// SIMATIC S7-200 project (STEP 7-Micro/WIN), CPU 226 CN REL 02.01

SYMBOL_TABLE 变量
接收字节数            VB0
从站地址             VB1
保持寄存器起始地址        VD2
最大IO点数           VW6
最大AI通道数          VW8      // 可为16或32
保持寄存器数量          VW10
数据包合法性           V12.0    // 只有该位为1才会处理数据包
接收存储区            VB13
发送存储区            VB268
END_SYMBOL_TABLE

SYMBOL_TABLE Modbus地址
M0001            QB0      // 00001~00128
M10001           IB0      // I0.0~I15.7
M3000            AIW0     // AIW0~AIW62
END_SYMBOL_TABLE

ORGANIZATION_BLOCK 主程序:OB1
TITLE=程序注释
BEGIN
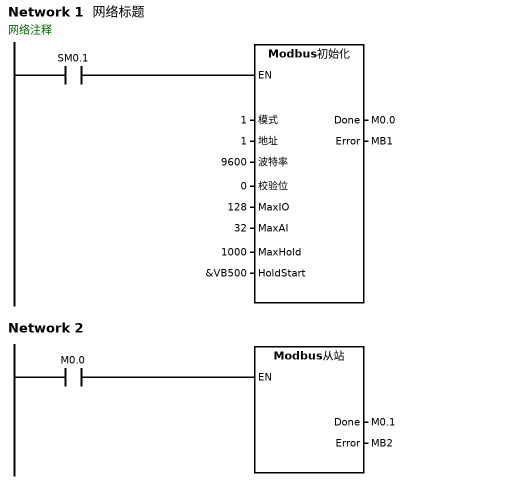
Network 1 // 网络标题
// 网络注释
LD     SM0.1
CALL   Modbus初始化:SBR0, 1, 1, 9600, 0, 128, 32, 1000, &VB500, M0.0, MB1
Network 2
LD     M0.0
CALL   Modbus从站:SBR1, M0.1, MB2
END_ORGANIZATION_BLOCK

SUBROUTINE_BLOCK Modbus初始化:SBR0
TITLE=此程序初始化Modbus所需参数
// 校验位:
// 0 - 无校验
// 1 - 奇校验
// 2 - 偶校验
// 
// Error值在Done位为0时有效
// Error值含义:
// 1 - 波特率初始化失败
// 2 - 校验位初始化失败
// 3 - 没有相关模式
VAR_INPUT
模式:BYTE;	// LB0 0 - 禁用Modbus库、1 - 启用Modbus库
地址:BYTE;	// LB1 从站地址
波特率:DWORD;	// LD2 通讯所需波特率
校验位:BYTE;	// LB6 数据包校验位
MaxIO:INT;	// LW7 
MaxAI:INT;	// LW9 可为16或32
MaxHold:INT;	// LW11 
HoldStart:DWORD;	// LD13 
END_VAR
VAR_OUTPUT
Done:BOOL;	// L17.0 0 - 初始化失败、1 - 初始化成功
Error:BYTE;	// LB18 
END_VAR
VAR
自由口控制:BYTE;	// LB19 
初始化标志:BYTE;	// LB20 
END_VAR
BEGIN
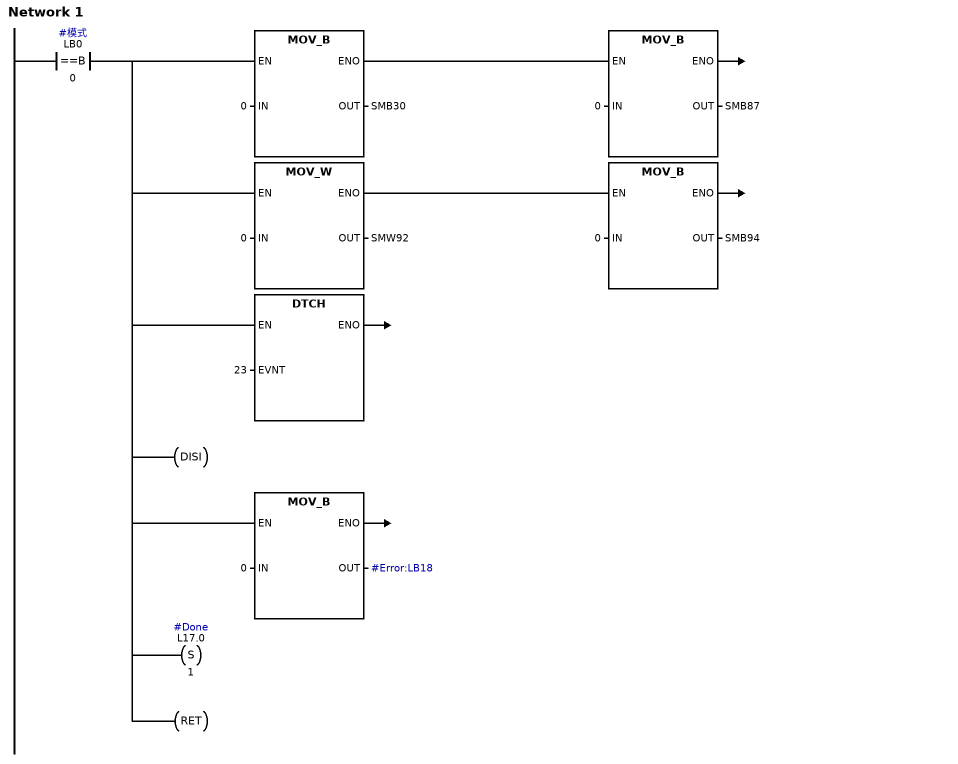
Network 1
LDB=   #模式:LB0, 0
LPS
MOVB   0, SMB30
AENO
MOVB   0, SMB87
LRD
MOVW   0, SMW92
AENO
MOVB   0, SMB94
LRD
DTCH   23
LRD
DISI
LRD
MOVB   0, #Error:LB18
LRD
S      #Done:L17.0, 1
LPP
CRET
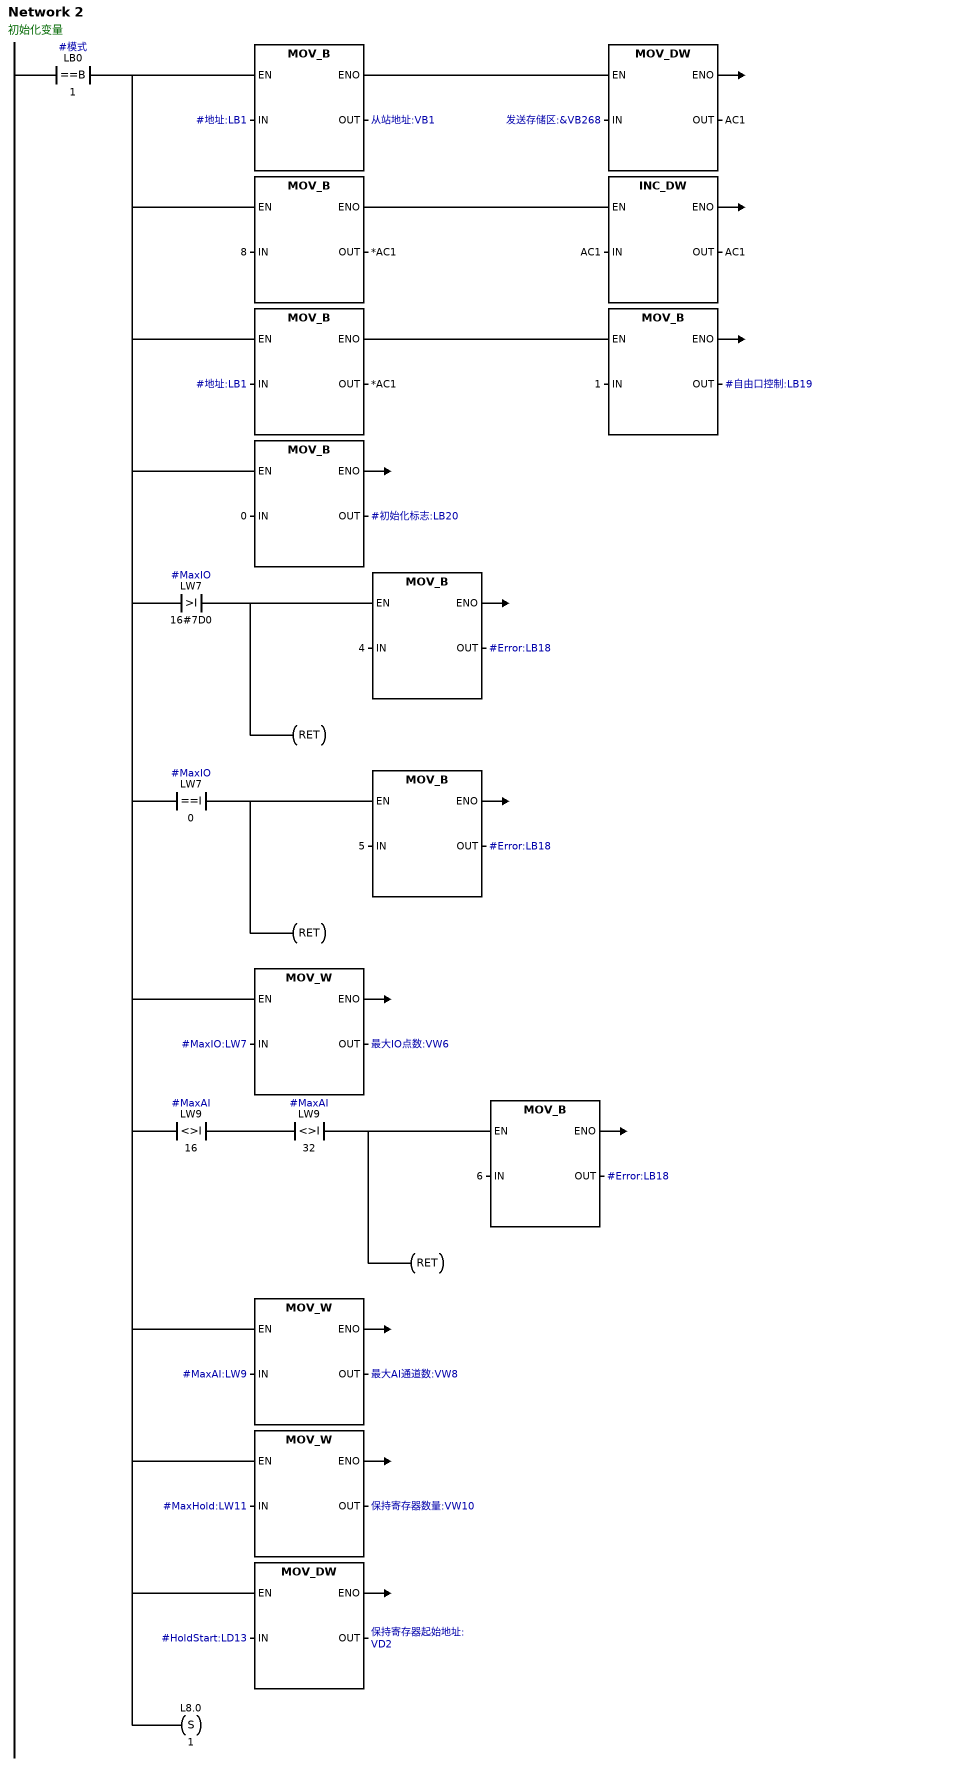
Network 2
// 初始化变量
LDB=   #模式:LB0, 1
LPS
MOVB   #地址:LB1, 从站地址:VB1
AENO
MOVD   &发送存储区:VB268, AC1
LRD
MOVB   8, *AC1
AENO
INCD   AC1
LRD
MOVB   #地址:LB1, *AC1
AENO
MOVB   1, #自由口控制:LB19
LRD
MOVB   0, #初始化标志:LB20
LRD
AW>    #MaxIO:LW7, 16#7D0
MOVB   4, #Error:LB18
CRET
LRD
AW=    #MaxIO:LW7, 0
MOVB   5, #Error:LB18
CRET
LRD
MOVW   #MaxIO:LW7, 最大IO点数:VW6
LRD
AW<>   #MaxAI:LW9, 16
AW<>   #MaxAI:LW9, 32
MOVB   6, #Error:LB18
CRET
LPP
MOVW   #MaxAI:LW9, 最大AI通道数:VW8
MOVW   #MaxHold:LW11, 保持寄存器数量:VW10
MOVD   #HoldStart:LD13, 保持寄存器起始地址:VD2
S      L8.0, 1
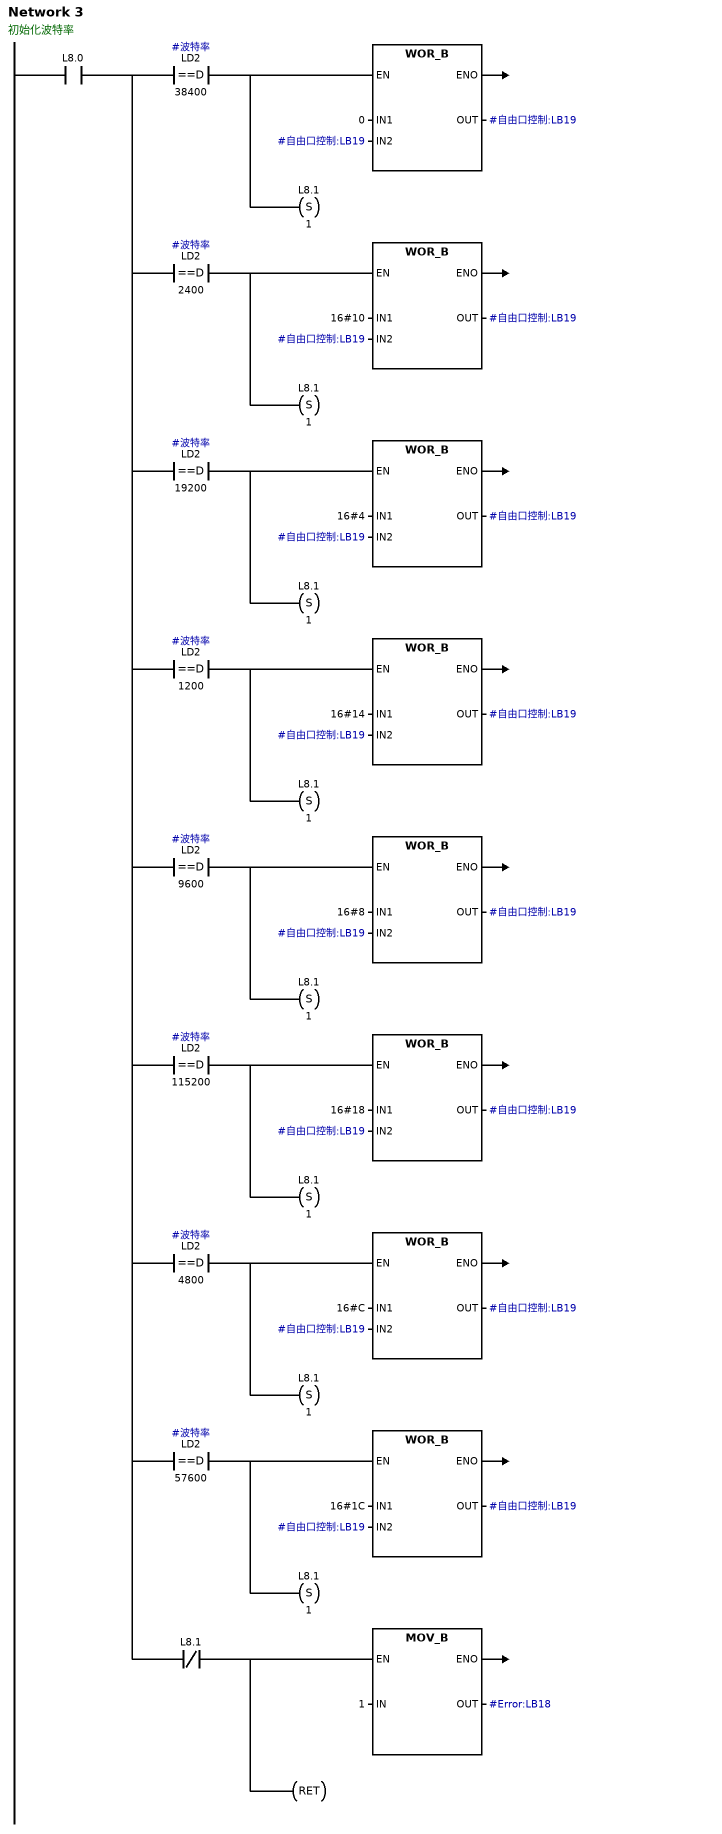
Network 3
// 初始化波特率
LD     L8.0
LPS
AD=    #波特率:LD2, 38400
ORB    0, #自由口控制:LB19
S      L8.1, 1
LRD
AD=    #波特率:LD2, 2400
ORB    16#10, #自由口控制:LB19
S      L8.1, 1
LRD
AD=    #波特率:LD2, 19200
ORB    16#4, #自由口控制:LB19
S      L8.1, 1
LRD
AD=    #波特率:LD2, 1200
ORB    16#14, #自由口控制:LB19
S      L8.1, 1
LRD
AD=    #波特率:LD2, 9600
ORB    16#8, #自由口控制:LB19
S      L8.1, 1
LRD
AD=    #波特率:LD2, 115200
ORB    16#18, #自由口控制:LB19
S      L8.1, 1
LRD
AD=    #波特率:LD2, 4800
ORB    16#C, #自由口控制:LB19
S      L8.1, 1
LRD
AD=    #波特率:LD2, 57600
ORB    16#1C, #自由口控制:LB19
S      L8.1, 1
LPP
AN     L8.1
MOVB   1, #Error:LB18
CRET
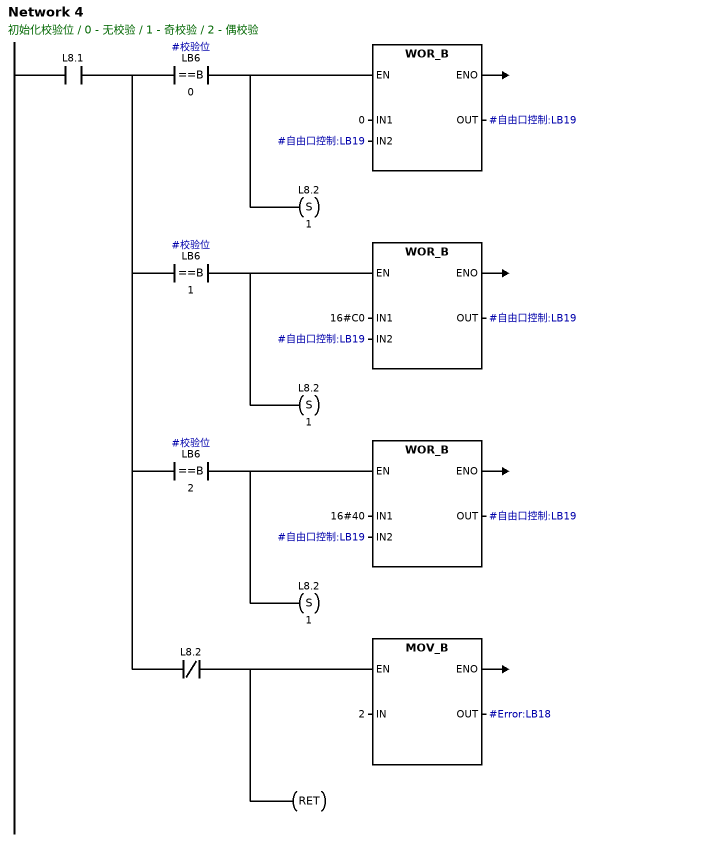
Network 4
// 初始化校验位
// 0 - 无校验
// 1 - 奇校验
// 2 - 偶校验
LD     L8.1
LPS
AB=    #校验位:LB6, 0
ORB    0, #自由口控制:LB19
S      L8.2, 1
LRD
AB=    #校验位:LB6, 1
ORB    16#C0, #自由口控制:LB19
S      L8.2, 1
LRD
AB=    #校验位:LB6, 2
ORB    16#40, #自由口控制:LB19
S      L8.2, 1
LPP
AN     L8.2
MOVB   2, #Error:LB18
CRET
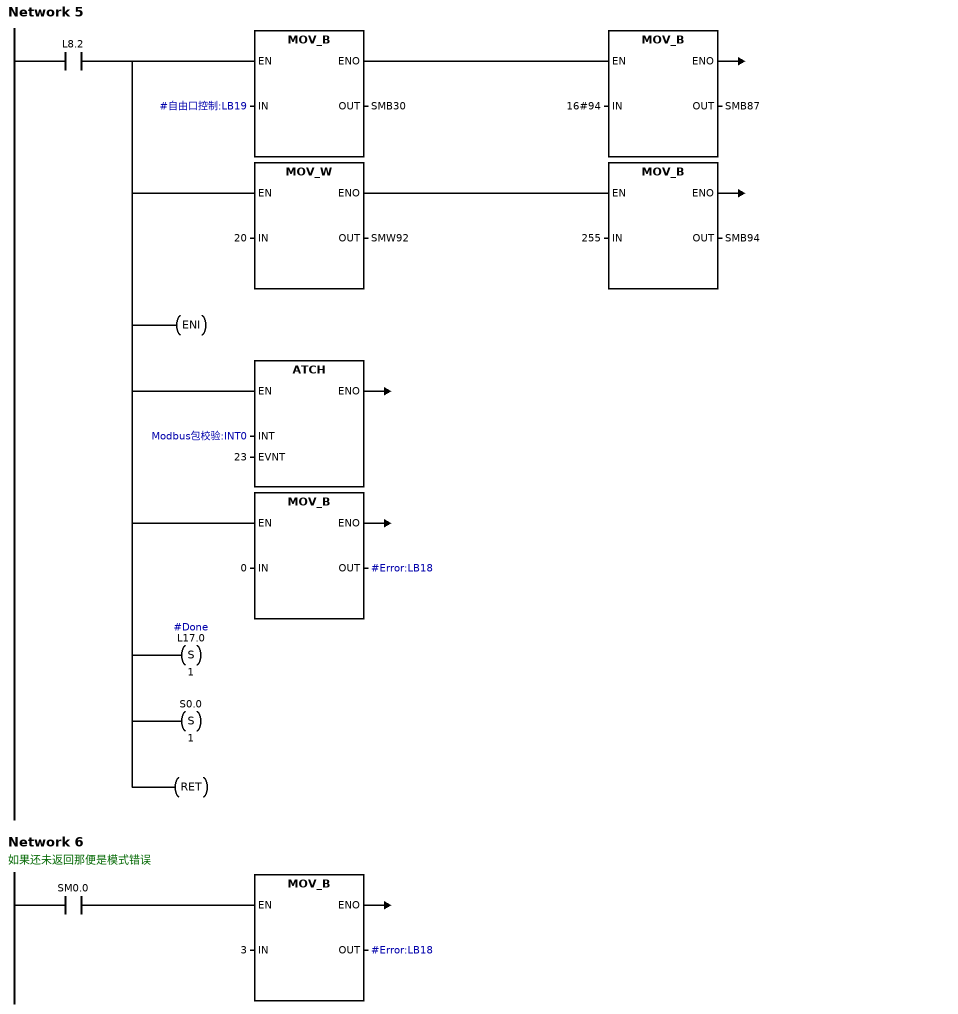
Network 5
LD     L8.2
LPS
MOVB   #自由口控制:LB19, SMB30
AENO
MOVB   16#94, SMB87
LRD
MOVW   20, SMW92
AENO
MOVB   255, SMB94
LRD
ENI
LRD
ATCH   Modbus包校验:INT0, 23
LRD
MOVB   0, #Error:LB18
LRD
S      #Done:L17.0, 1
LRD
S      S0.0, 1
LPP
CRET
Network 6
// 如果还未返回那便是模式错误
LD     SM0.0
MOVB   3, #Error:LB18
END_SUBROUTINE_BLOCK

SUBROUTINE_BLOCK Modbus从站:SBR1
TITLE=该子程序解析并处理数据包,同时也会构建回复包返回
// 需要使用STL代码编辑器查看
// 
// AC1 - 地址区指针
// AC2 - 数据区指针
// AC3 - 通用指针
// 
// 当跳转至具体功能执行前:
// * AC1将指向接收存储区的地址区
// * AC2将指向接收存储区的功能码区
// * AC3将指向发送区首地址+2 (跳过包头和从站地址)
VAR_OUTPUT
Done:BOOL;	// L0.0 0 - 空闲状态、1 - 正在处理数据
Error:BYTE;	// LB1 和Modbus协议中异常码一致
END_VAR
VAR
功能码:BYTE;	// LB2 
地址:DWORD;	// LD3 
数据数量:WORD;	// LW7 
通用存储B:BYTE;	// LB9 
通用存储B2:BYTE;	// LB10 
通用存储W:WORD;	// LW11 
通用存储W2:WORD;	// LW13 
通用存储W3:WORD;	// LW15 
通用存储D:DWORD;	// LD17 
通用存储D2:DWORD;	// LD21 
END_VAR
BEGIN
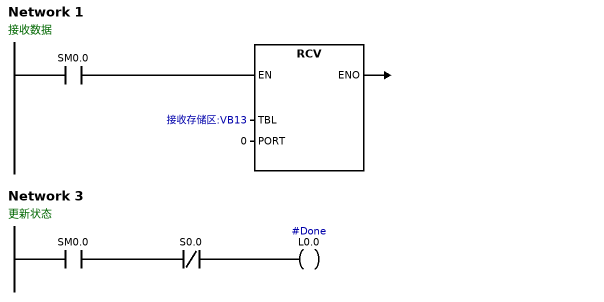
Network 1
// 接收数据
LD     SM0.0
RCV    接收存储区:VB13, 0
Network 2
// 功能码判断
// 通过段转移的方式能保证在执行完当前功能前不处理任何其它请求以防止冲突
LSCR   S0.0
LD     SM0.0
MOVB   0, #Error:LB1
LD     数据包合法性:V12.0
LPS
MOVD   &接收存储区:VB13, AC1
AENO
+D     3, AC1
LRD
MOVD   &接收存储区:VB13, AC2
AENO
+D     2, AC2
LRD
MOVD   &发送存储区:VB268, AC3
AENO
+D     2, AC3
LRD
AB=    *AC2, 1
MOVB   1, #功能码:LB2
MOVD   &M0001:QB0, #地址:LD3
SCRT   S0.1
?32B
LRD
AB=    *AC2, 2
MOVB   2, #功能码:LB2
MOVD   &M10001:IB0, #地址:LD3
SCRT   S0.1
?32B
LRD
AB=    *AC2, 3
MOVB   3, #功能码:LB2
MOVD   保持寄存器起始地址:VD2, #地址:LD3
SCRT   S0.2
?32B
LRD
AB=    *AC2, 4
MOVB   4, #功能码:LB2
MOVD   &M3000:AIW0, #地址:LD3
SCRT   S0.2
?32B
LRD
AB=    *AC2, 5
SCRT   S0.3
?32B
LRD
AB=    *AC2, 6
SCRT   S0.4
?32B
LRD
AB=    *AC2, 15
SCRT   S0.5
?32B
LRD
AB=    *AC2, 16
SCRT   S0.6
?32B
LPP
CALL   发送出错包:SBR4, 1
MOVB   1, #Error:LB1
SCRE
Network 3
// 更新状态
LD     SM0.0
AN     S0.0
=      #Done:L0.0
Network 4
// 01H & 02H
LSCR   S0.1
LD     SM0.0
LPS
A      SM1.1
CALL   发送出错包:SBR4, 4
MOVB   4, #Error:LB1
LRD
+D     3, AC2
AENO
MOVW   *AC2, #数据数量:LW7
/I     +8, #数据数量:LW7
LRD
LDW=   *AC2, 0
OW>    *AC2, 最大IO点数:VW6
ALD
CALL   发送出错包:SBR4, 3
MOVB   3, #Error:LB1
SCRT   S0.0
?32B
LRD
MOVW   *AC1, #通用存储W2:LW13
+I     *AC2, #通用存储W2:LW13
LRD
LDW>   *AC1, 16#7D0
OW>    #通用存储W2:LW13, 16#7D0
ALD
CALL   发送出错包:SBR4, 2
MOVB   2, #Error:LB1
SCRT   S0.0
?32B
LPP
LPS
MOVW   #数据数量:LW7, #通用存储W:LW11
AENO
*I     +8, #通用存储W:LW11
AENO
INVW   #通用存储W:LW11
INCW   #通用存储W:LW11
+I     *AC2, #通用存储W:LW11
LRD
AW<>   #通用存储W:LW11, 0
INCW   #数据数量:LW7
LRD
MOVD   #地址:LD3, AC2
AENO
ITD    *AC1, #通用存储D:LD17
LRD
+D     #通用存储D:LD17, AC2
AENO
MOVB   #功能码:LB2, *AC3
LRD
INCD   AC3
AENO
ITB    #数据数量:LW7, *AC3
LRD
INCD   AC3
AENO
ITB    #数据数量:LW7, #通用存储B:LB9
LRD
BMB    *AC2, *AC3, #通用存储B:LB9
AENO
ITD    #数据数量:LW7, #通用存储D:LD17
LRD
+D     #通用存储D:LD17, AC3
MOVW   #数据数量:LW7, #通用存储W2:LW13
AENO
+I     +5, #通用存储W2:LW13
AENO
ITB    #通用存储W2:LW13, 发送存储区:VB268
LRD
AW<>   #通用存储W:LW11, 0
LPS
INVW   #通用存储W:LW11
AENO
INCW   #通用存储W:LW11
AENO
+I     8, #通用存储W:LW11
AENO
ITB    #通用存储W:LW11, #通用存储B:LB9
LRD
MOVB   16#FF, #通用存储B2:LB10
AENO
SRB    #通用存储B2:LB10, #通用存储B:LB9
AENO
DECD   AC3
LPP
ANDB   #通用存储B2:LB10, *AC3
LPP
CALL   发送数据包:SBR3
SCRT   S0.0
SCRE
Network 5
// 03H & 04H
LSCR   S0.2
LD     SM0.0
LPS
A      SM1.1
CALL   发送出错包:SBR4, 4
MOVB   4, #Error:LB1
SCRT   S0.0
?32B
LRD
+D     3, AC2
AENO
MOVW   *AC2, #数据数量:LW7
LRD
LDW=   #数据数量:LW7, 0
LDB=   #功能码:LB2, 3
AW>    #数据数量:LW7, 保持寄存器数量:VW10
OLD
LDB=   #功能码:LB2, 4
AW>    #数据数量:LW7, 最大AI通道数:VW8
OLD
ALD
CALL   发送出错包:SBR4, 3
MOVB   3, #Error:LB1
SCRT   S0.0
?32B
LRD
MOVW   *AC1, #通用存储W:LW11
+I     #数据数量:LW7, #通用存储W:LW11
LRD
LDW>   *AC1, 保持寄存器数量:VW10
OW>    #通用存储W:LW11, 保持寄存器数量:VW10
ALD
CALL   发送出错包:SBR4, 2
MOVB   2, #Error:LB1
SCRT   S0.0
?32B
LPP
LPS
MOVD   #地址:LD3, AC2
AENO
ITD    *AC1, #通用存储D2:LD21
LRD
*D     2, #通用存储D2:LD21
AENO
+D     #通用存储D2:LD21, AC2
LRD
MOVB   #功能码:LB2, *AC3
AENO
INCD   AC3
LRD
MOVW   #数据数量:LW7, #通用存储W:LW11
AENO
*I     +2, #通用存储W:LW11
AENO
ITB    #通用存储W:LW11, *AC3
LRD
INCD   AC3
AENO
ITB    #数据数量:LW7, #通用存储B:LB9
LRD
BMW    *AC2, *AC3, #通用存储B:LB9
*I     2, #数据数量:LW7
AENO
MOVW   #数据数量:LW7, #通用存储W:LW11
+I     +5, #通用存储W:LW11
LRD
ITB    #通用存储W:LW11, 发送存储区:VB268
AENO
CALL   发送数据包:SBR3
LPP
SCRT   S0.0
SCRE
Network 6
// 05H
// AC1 - 通用指针
// AC2 - 协议数据区地址
// AC3 - S7-200数据区地址
LSCR   S0.3
LD     SM0.0
LPS
MOVW   最大IO点数:VW6, #通用存储W:LW11
-I     1, #通用存储W:LW11
AW>    *AC1, #通用存储W:LW11
CALL   发送出错包:SBR4, 2
MOVB   2, #Error:LB1
SCRT   S0.0
?32B
LRD
LPS
MOVW   *AC1, #通用存储W:LW11
AENO
/I     +8, #通用存储W:LW11
AENO
MOVD   &M0001:QB0, AC3
LRD
ITD    #通用存储W:LW11, #通用存储D:LD17
AENO
+D     #通用存储D:LD17, AC3
LRD
AW<>   #通用存储W:LW11, 0
*I     8, #通用存储W:LW11
LRD
INVW   #通用存储W:LW11
AENO
INCW   #通用存储W:LW11
AENO
+I     *AC1, #通用存储W:LW11
AENO
ITB    #通用存储W:LW11, #通用存储B:LB9
LRD
MOVB   1, #通用存储B2:LB10
AENO
SLB    #通用存储B2:LB10, #通用存储B:LB9
AENO
+D     3, AC2
LPP
AW=    *AC2, 16#FF00
ORB    #通用存储B2:LB10, *AC3
LRD
AW=    *AC2, 0
INVB   #通用存储B2:LB10
ANDB   #通用存储B2:LB10, *AC3
LPP
AW<>   *AC2, 16#FF00
AW<>   *AC2, 0
CALL   发送出错包:SBR4, 3
MOVB   3, #Error:LB1
SCRT   S0.0
?32B
LPP
LPS
LD     SM1.1
CALL   发送出错包:SBR4, 4
MOVB   4, #Error:LB1
SCRT   S0.0
?32B
LPP
MOVB   8, 接收存储区:VB13
SCPY   接收存储区:VB13, 发送存储区:VB268
CALL   发送数据包:SBR3
SCRT   S0.0
SCRE
Network 7
// 06H
// AC1 - 通用指针
// AC2 - 协议数据区地址
// AC3 - S7-200数据区地址
// 
// 寄存器的值将永远不会超出范围,所以错误码3将被忽略以提升性能
LSCR   S0.4
LD     SM0.0
LPS
MOVD   保持寄存器起始地址:VD2, AC3
AENO
MOVW   *AC1, #通用存储W:LW11
*I     +2, #通用存储W:LW11
LRD
MOVW   保持寄存器数量:VW10, #通用存储W2:LW13
*I     +2, #通用存储W2:LW13
LRD
AW>    *AC1, #通用存储W2:LW13
CALL   发送出错包:SBR4, 2
MOVB   2, #Error:LB1
SCRT   S0.0
?32B
LPP
LPS
ITD    #通用存储W:LW11, #通用存储D:LD17
AENO
+D     #通用存储D:LD17, AC3
LPP
+D     +3, AC2
AENO
MOVW   *AC2, *AC3
LPS
LD     SM1.1
CALL   发送出错包:SBR4, 4
MOVB   4, #Error:LB1
SCRT   S0.0
?32B
LPP
MOVB   8, 接收存储区:VB13
SCPY   接收存储区:VB13, 发送存储区:VB268
CALL   发送数据包:SBR3
SCRT   S0.0
SCRE
Network 8
// 0FH
LSCR   S0.5
LD     SM0.0
LPS
+D     +3, AC2
AENO
MOVW   *AC2, #通用存储W:LW11
LRD
+D     +2, AC2
AENO
BTI    接收字节数:VB0, #通用存储W2:LW13
LRD
-I     +9, #通用存储W2:LW13
AENO
ITB    #通用存储W2:LW13, #通用存储B:LB9
LRD
MOVW   #通用存储W:LW11, #通用存储W3:LW15
AENO
/I     +8, #通用存储W3:LW15
AENO
*I     +8, #通用存储W3:LW15
LRD
LDW>   #通用存储W:LW11, 16#7B0
OW=    #通用存储W:LW11, +0
OB<>   #通用存储B:LB9, *AC2
OW<>   #通用存储W3:LW15, #通用存储W:LW11
ALD
CALL   发送出错包:SBR4, 3
MOVB   3, #Error:LB1
SCRT   S0.0
?32B
LRD
MOVW   #通用存储W:LW11, #通用存储W2:LW13
+I     *AC1, #通用存储W2:LW13
LRD
LDW>   *AC1, 保持寄存器数量:VW10
OW>    #通用存储W2:LW13, 保持寄存器数量:VW10
ALD
CALL   发送出错包:SBR4, 2
MOVB   2, #Error:LB1
SCRT   S0.0
?32B
LPP
LPS
/I     +8, #通用存储W:LW11
AENO
INCD   AC2
LRD
MOVD   &M0001:QB0, AC3
AENO
ITD    *AC1, #通用存储D:LD17
LRD
+D     #通用存储D:LD17, AC3
LRD
ITB    #通用存储W:LW11, #通用存储B:LB9
BMB    *AC2, *AC3, #通用存储B:LB9
LPP
LPS
LD     SM1.1
CALL   发送出错包:SBR4, 4
MOVB   4, #Error:LB1
SCRT   S0.0
?32B
LPP
LPS
MOVB   8, 接收存储区:VB13
AENO
SCPY   接收存储区:VB13, 发送存储区:VB268
LRD
MOVD   &发送存储区:VB268, AC1
AENO
+D     +6, AC1
LRD
CALL   发送数据包:SBR3
LPP
SCRT   S0.0
SCRE
Network 9
// 10H
LSCR   S0.6
LD     SM0.0
LPS
+D     +3, AC2
AENO
MOVW   *AC2, #通用存储W:LW11
LRD
BTI    接收字节数:VB0, #通用存储W2:LW13
AENO
-I     +9, #通用存储W2:LW13
LRD
+D     +2, AC2
AENO
ITB    #通用存储W2:LW13, #通用存储B:LB9
LRD
LDW>   #通用存储W:LW11, 16#7B0
OW=    #通用存储W:LW11, +0
OB<>   #通用存储B:LB9, *AC2
ALD
CALL   发送出错包:SBR4, 3
MOVB   3, #Error:LB1
SCRT   S0.0
?32B
LRD
MOVW   #通用存储W:LW11, #通用存储W2:LW13
+I     *AC1, #通用存储W2:LW13
LRD
LDW>   *AC1, 保持寄存器数量:VW10
OW>    #通用存储W2:LW13, 保持寄存器数量:VW10
ALD
CALL   发送出错包:SBR4, 2
MOVB   2, #Error:LB1
SCRT   S0.0
?32B
LPP
LPS
INCD   AC2
AENO
MOVD   保持寄存器起始地址:VD2, AC3
LRD
ITD    *AC1, #通用存储D:LD17
AENO
*D     +2, #通用存储D:LD17
LRD
+D     #通用存储D:LD17, AC3
LRD
ITB    #通用存储W:LW11, #通用存储B:LB9
BMW    *AC2, *AC3, #通用存储B:LB9
LPP
LPS
LD     SM1.1
CALL   发送出错包:SBR4, 4
MOVB   4, #Error:LB1
SCRT   S0.0
?32B
LPP
LPS
MOVB   8, 接收存储区:VB13
AENO
SCPY   接收存储区:VB13, 发送存储区:VB268
LRD
MOVD   &发送存储区:VB268, AC1
AENO
+D     +6, AC1
LRD
CALL   发送数据包:SBR3
LPP
SCRT   S0.0
SCRE
END_SUBROUTINE_BLOCK

SUBROUTINE_BLOCK Modbus_CRC16:SBR2
TITLE=该子程序计算CRC校验
VAR_INPUT
Start:DWORD;	// LD0 起始地址
Lenth:INT;	// LW4 长度
END_VAR
VAR_OUTPUT
CRC:INT;	// LW6 
END_VAR
VAR
CRC_Register:WORD;	// LW8 
For1:WORD;	// LW10 
For2:WORD;	// LW12 
END_VAR
BEGIN
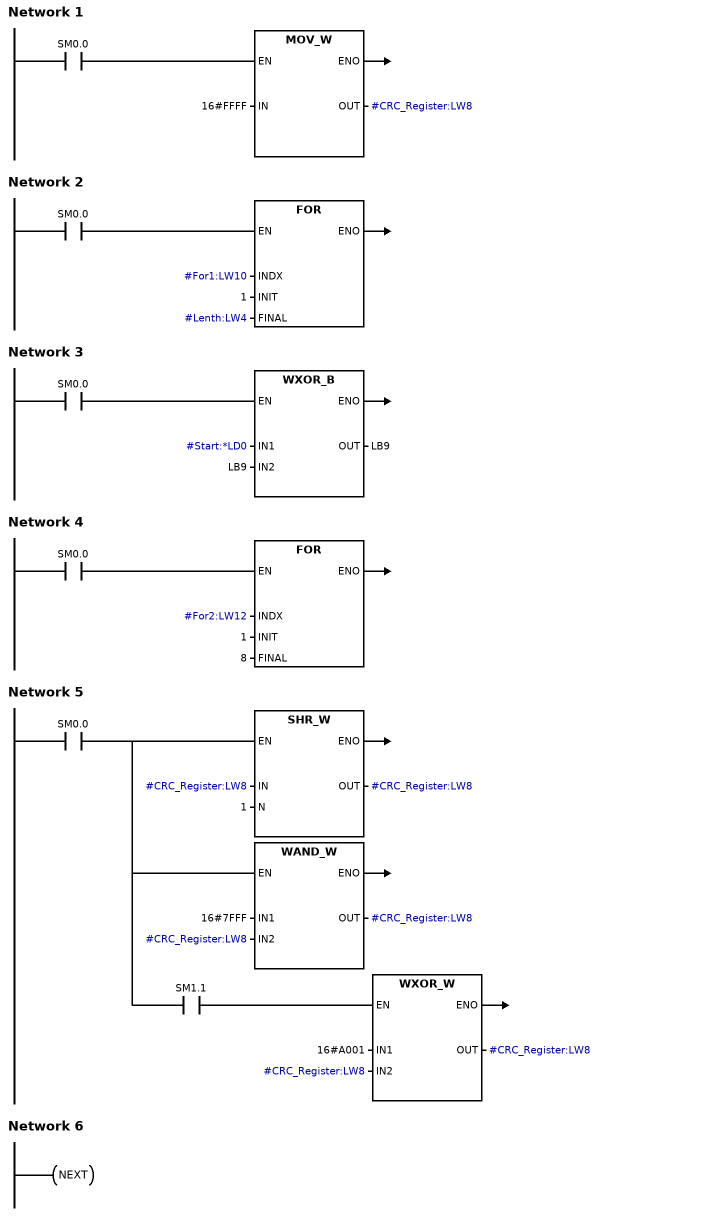
Network 1
LD     SM0.0
MOVW   16#FFFF, #CRC_Register:LW8
Network 2
LD     SM0.0
FOR    #For1:LW10, 1, #Lenth:LW4
Network 3
LD     SM0.0
XORB   *#Start:LD0, LB9
Network 4
LD     SM0.0
FOR    #For2:LW12, 1, 8
Network 5
LD     SM0.0
SRW    #CRC_Register:LW8, 1
ANDW   16#7FFF, #CRC_Register:LW8
A      SM1.1
XORW   16#A001, #CRC_Register:LW8
Network 6
NEXT
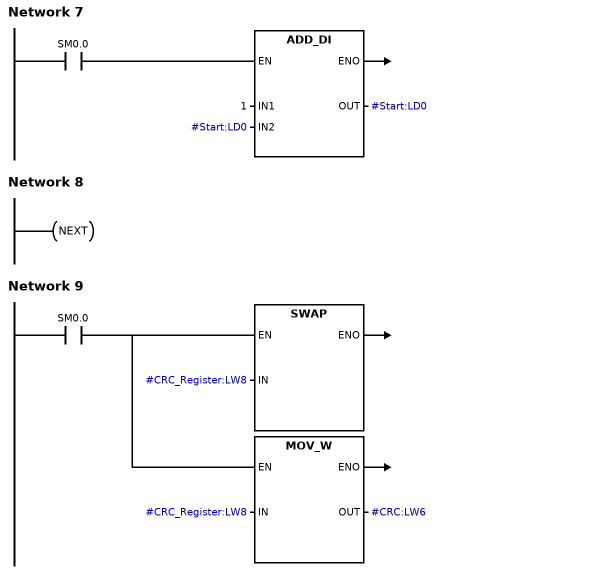
Network 7
LD     SM0.0
+D     1, #Start:LD0
Network 8
NEXT
Network 9
LD     SM0.0
SWAP   #CRC_Register:LW8
MOVW   #CRC_Register:LW8, #CRC:LW6
END_SUBROUTINE_BLOCK

SUBROUTINE_BLOCK 发送数据包:SBR3
TITLE=在数据包后添加CRC校验并发送出去
VAR
数据包包长度W:WORD;	// LW0 
数据包包长度D:DWORD;	// LD2 
END_VAR
BEGIN
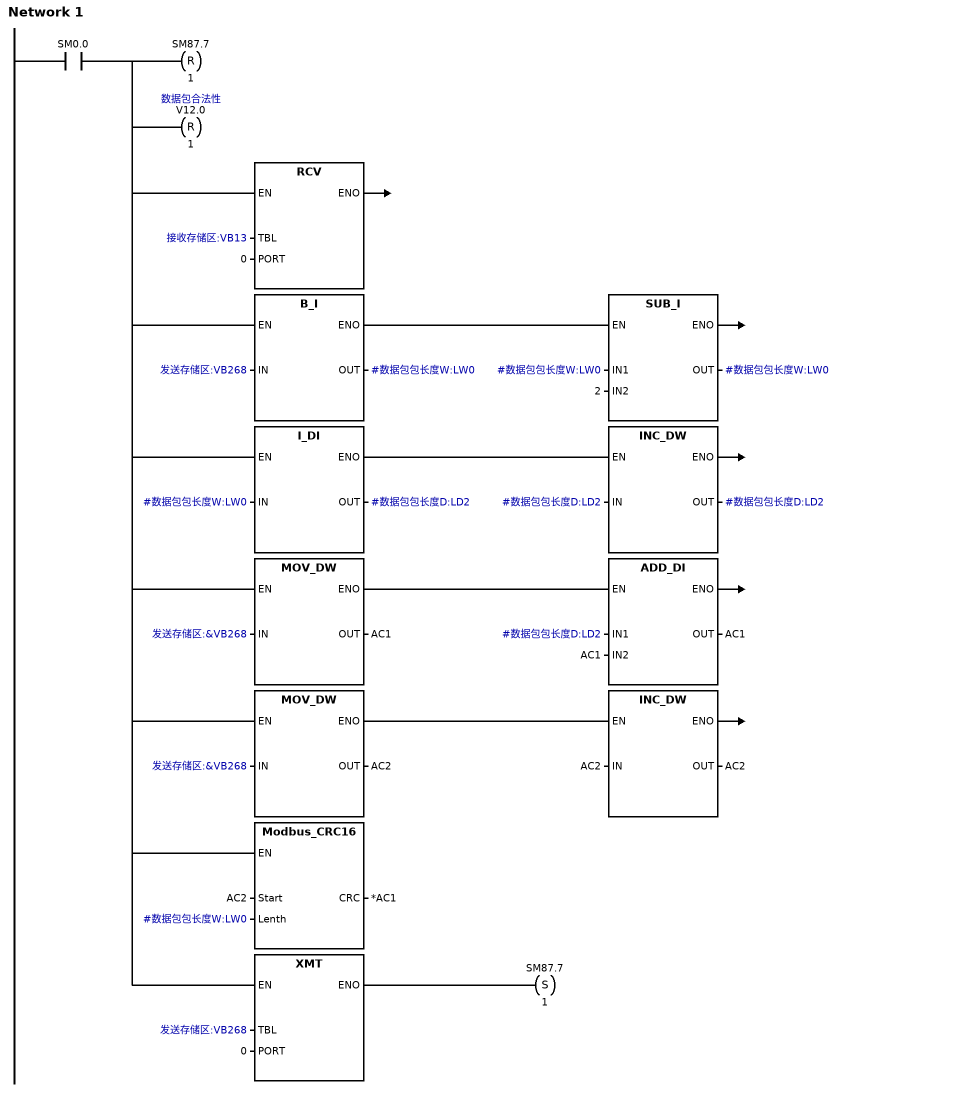
Network 1
LD     SM0.0
LPS
R      SM87.7, 1
R      数据包合法性:V12.0, 1
RCV    接收存储区:VB13, 0
BTI    发送存储区:VB268, #数据包包长度W:LW0
AENO
-I     2, #数据包包长度W:LW0
LRD
ITD    #数据包包长度W:LW0, #数据包包长度D:LD2
AENO
INCD   #数据包包长度D:LD2
LRD
MOVD   &发送存储区:VB268, AC1
AENO
+D     #数据包包长度D:LD2, AC1
LRD
MOVD   &发送存储区:VB268, AC2
AENO
INCD   AC2
LRD
CALL   Modbus_CRC16:SBR2, AC2, #数据包包长度W:LW0, *AC1
LPP
XMT    发送存储区:VB268, 0
AENO
S      SM87.7, 1
END_SUBROUTINE_BLOCK
